// TIA Portal V20 export
// export: Created 2025-12-01T14:57:12.7432342Z, ExportSetting None, DisplayName Totally Integrated Automation Portal, DisplayVersion V20 Update 3, DisplayName TIA Portal Openness, DisplayVersion V20 Update 3, DisplayName TIA Portal Version Control Interface, DisplayVersion V20 Update 3, DisplayName STEP 7 Professional, DisplayVersion V20 Update 3, DisplayName STEP 7 Safety, DisplayVersion V20 Update 2, DisplayName WinCC Basic/Comfort/Advanced, DisplayVersion V20 Update 3, DisplayName WinCC Professional, DisplayVersion V20 Update 3, DisplayName WinCC Unified, DisplayVersion V20 Update 3
FUNCTION "FC756_EventosEstadoProcesoMaquina" : Void   // FC756, STL
TITLE = Emision de los Eventos del Proceso de la Maquina
{ S7_Optimized_Access := 'FALSE' }
AUTHOR : TRACKING
NAME : 20141014
VERSION : 4.0
// stored: AutoNumber false
   VAR_INPUT
      NumMaquina : UInt;   // Numero de Maquina
      EstadoMaquina : "EstadoZona";   // Estado de la Maquina
      EstadoVIMaquina : "EstadoMaquina";   // Estado del VI de la Maquina
      EmpezandoProceso : Bool;   // Aviso de Empezando el Proceso
      FinalProceso : Bool;   // Aviso de Final del Proceso
      ErrorProceso : Bool;   // Aviso de Error de Proceso
      MesaDeJDT02 : Bool;
   END_VAR
   VAR_TEMP
      NumeroUT : UInt;
      ProcesoActual : UInt;
      P_EmiEventos : DWord;
      DBEventos : Word;
      NumDBEventos : UInt;
      MaxBytes : UInt;
      NumBytes : UInt;
      OffsetInicial : UInt;
      OffsetFinal : UInt;
      Conversion : DWord;
      Convertir : UInt;
      Valor : UDInt;
   END_VAR
BEGIN

NETWORK
TITLE = Inicializaciones
///////////////////////////////////////////////////////////////////////////////
/// Inicio --> Pertenece al JDT 02

      L     "JDT1_NDB_EventosEmi";
      T     #DBEventos;
      T     #NumDBEventos;
      L     "JDT1_MaxBytes";
      T     #MaxBytes;

      AN    #MesaDeJDT02;
      JC    NoJdT02;

      L     "JDT2_NDB_EventosEmi";
      T     #DBEventos;
      T     #NumDBEventos;
      L     "JDT2_MaxBytes";
      T     #MaxBytes;

NoJdT02:NOP   0;

/// Final --> Pertenece al JDT 02
///////////////////////////////////////////////////////////////////////////////



NETWORK
TITLE = Mirar si se pueden generar eventos
// - Inicializo el Numero de Bytes y el puntero del DB de Eventos Generados
// - Calcula el Tamaño de bytes que hay en el DB de Eventos Genardos
// - Comprobamos si hay sitio para Eventos
///////////////////////////////////////////////////////////////////////////////
// Inicializo el Numero de Bytes y el puntero del DB Eventos Generados

      L     0;
      T     #NumBytes;  // Inicializo el numero de Bytes
      LAR2;  // Inicializo el puntero de Eventos Generados

///////////////////////////////////////////////////////////////////////////////
// Calcula el tamaño de bytes que hay en el DB Eventos Generados

      OPN   DB [#DBEventos];

Inicio_BusquedaFinalEventos:NOP   0;
      L     DBB [AR2, P#0.0];
      L     0;
      ==I;
      JC    Final_BusquedaFinalEventos;  // Buscamos el final del DB = 0

      +AR2  P#1.0;
      JU    Inicio_BusquedaFinalEventos;

Final_BusquedaFinalEventos:NOP   0;
      TAR2;  // Guardo el puntero
      T     #P_EmiEventos;  // Sacamos el NumBytes Escritos
      SRD   3;
      T     #NumBytes;

// -----------------------------------------------------------------------------------------------
// Comprobamos si hay sitio para mas Eventos

      L     #NumBytes;  // Miramos si hay sitio
      L     #MaxBytes;  // Max. que se pueden emitir, parametro
      >I;
      JC    Final;  // No se pueden generar más eventos



NETWORK
TITLE = Distribucion
///////////////////////////////////////////////////////////////////////////////
// --- Distribucion  del Estado del Proceso de la Maquina

      L     0;
      T     #ProcesoActual;

// ---------- Mirar si el Proceso esta Empezando

      A     #EmpezandoProceso;
      AN    #FinalProceso;
      AN    #ErrorProceso;
      JCN   _ST1;  // No Esta Empezando ?

      L     1011;  // Esta Empezando
      T     #ProcesoActual;
      JU    _STF;


// ---------- Mirar si el Proceso ha Finalizado

_ST1: AN    #EmpezandoProceso;
      A     #FinalProceso;
      AN    #ErrorProceso;
      JCN   _ST2;  // No Esta Finalizado ?

      L     1012;  // Esta Finalizado
      T     #ProcesoActual;
      JU    _STF;


// ---------- Mirar si el Proceso esta en Error

_ST2: AN    #EmpezandoProceso;
      AN    #FinalProceso;
      A     #ErrorProceso;
      JCN   _ST3;  // No Esta En Error ?

      L     1013;  // Esta En Error
      T     #ProcesoActual;
      JU    _STF;


// ---------- No se sabe como esta el Proceso

_ST3: L     0;  // No se Sabe
      T     "DB832_Maquinas".Maquinas[#NumMaquina].MemoriaEstado;  // Guardo como Nuevo

      JU    ST_F;


///////////////////////////////////////////////////////////////////////////////
// ---------- Mirar si hay que Emitir el Evento

_STF: NOP   0;
      L     "DB832_Maquinas".Maquinas[#NumMaquina].MemoriaEstado;
      L     #ProcesoActual;
      ==I;
      JC    ST_F;  // No ha cambio de Proceso ?

      L     0;
      L     #ProcesoActual;
      ==I;
      JC    ST_F;  // Y no sea Indetermiado ?

      JU    EmitirEvento;


///////////////////////////////////////////////////////////////////////////////
// --- Fin del Control

ST_F: JU    Final;



NETWORK
TITLE = Emision del Evento
EmitirEvento:NOP   0;

///////////////////////////////////////////////////////////////////////////////
// --- Formateo del Evento PROC - Estado del Proceso de la Maquina

      L     #P_EmiEventos;
      LAR2;  // Puntero al DB de Eventos Generados

      TAR2;  // Mirar si es el primer evento de la lista
      L     0;
      ==I;
      JC    NoEsInicio_ListaDeEventos;  // Es el primero

      OPN   DB [#DBEventos];
      L     ',';  // Separador entre eventos ','
      T     DBB [AR2, P#0.0];
      +AR2  P#1.0;

NoEsInicio_ListaDeEventos:NOP   0;
      OPN   DB [#DBEventos];  // DB de Eventos Generados (A Emitir)
      L     '{';  // Inicio de Evento '{'
      T     DBB [AR2, P#0.0];
      +AR2  P#1.0;


///////////////////////////////////////////////////////////////////////////////
// --- Cuerpo del Evento PROC

      L     'DATO';  // Evento 'DATO'
      T     DBD [AR2, P#0.0];
      +AR2  P#4.0;

      L     '[';  // Evento - Atributo Proceso '[PROC]'
      T     DBB [AR2, P#0.0];
      L     'PROC';
      T     DBD [AR2, P#1.0];
      L     ']';
      T     DBB [AR2, P#5.0];
      +AR2  P#6.0;

      L     "DB850_DefinicionMesas".Mesa[#NumMaquina].ConfigMesa.TipoMaquina;
      T     #Convertir;

      CALL  "FC895_Obtener_EtiquetaDeValor"
      ( ValorEvento    := #Convertir,
        EtiquetaEvento := #Conversion
      );

      OPN   DB [#DBEventos];
      L     #Conversion;
      T     DBD [AR2, P#0.0];
      +AR2  P#4.0;

      L     '[';  // Evento - Atributo MCKY '[MCKY]'
      T     DBB [AR2, P#0.0];
      L     'MCKY';
      T     DBD [AR2, P#1.0];
      L     ']';
      T     DBB [AR2, P#5.0];
      +AR2  P#6.0;

      TAR2;  // Guardar el Puntero
      T     #P_EmiEventos;  // Al DB de Eventos Generados

// --- Obtener Numero de McKey

      L     "DB810_ColasMesas".Colas[#NumMaquina].UT_PrimeraMesa;
      T     #NumeroUT;

      L     "DB812_UTs_Control".UT[#NumeroUT].Mckey;
      T     #Valor;

// --- Fin de Obtener el Mckey

      L     #P_EmiEventos;  // Recuperar el Puntero
      LAR2;  // Al DB de Eventos Generados

// --- Convertir Valor a ASCII - Mckey
      TAR2;
      SRD   3;
      T     #OffsetInicial;  // Miro que offset tiene la String

      CALL  "FC893_Obtener_StringDelAtributo"
      ( DB_String := #NumDBEventos,
        OffsetIni := #OffsetInicial,
        Valor     := #Valor,
        OffsetFin := #OffsetFinal
      );  // Llamo a ObtenerStrinAtributo

      L     #OffsetFinal;
      SLD   3;
      LAR2;  // Recupero que offset tiene la String

// --- Ya esta convertido el Valor a ASCI - Fin Mckey

      OPN   DB [#DBEventos];  // DB de Eventos Generados (A Emitir)
      L     '[';  // Evento - Atributo MESA '[MESA]'
      T     DBB [AR2, P#0.0];
      L     'MESA';
      T     DBD [AR2, P#1.0];
      L     ']';
      T     DBB [AR2, P#5.0];
      +AR2  P#6.0;

// --- Convertir Valor a ASCII - Numero de Mesa
      TAR2;
      SRD   3;
      T     #OffsetInicial;  // Miro que offset tiene la String

      L     "CTE_OffsetMesa";
      L     #NumMaquina;  // Numero de Maquina
      +I;
      T     #Valor;

      CALL  "FC893_Obtener_StringDelAtributo"
      ( DB_String := #NumDBEventos,
        OffsetIni := #OffsetInicial,
        Valor     := #Valor,
        OffsetFin := #OffsetFinal
      );  // Llamo a ObtenerStrinAtributo

      L     #OffsetFinal;
      SLD   3;
      LAR2;  // Recupero que offset tiene la String

// --- Ya esta convertido el Valor a ASCI - Numero de Mesa

      OPN   DB [#DBEventos];  // DB de Eventos Generados (A Emitir)
      L     '[';  // Evento - Atributo Resultado '[RSLT]'
      T     DBB [AR2, P#0.0];
      L     'RSLT';
      T     DBD [AR2, P#1.0];
      L     ']';
      T     DBB [AR2, P#5.0];
      +AR2  P#6.0;

      L     #ProcesoActual;
      T     #Convertir;  // Proceso _INI o _FIN o ERRO

      CALL  "FC895_Obtener_EtiquetaDeValor"
      ( ValorEvento    := #Convertir,
        EtiquetaEvento := #Conversion
      );

      OPN   DB [#DBEventos];  // DB de Eventos Generados (A Emitir)
      L     #Conversion;
      T     DBD [AR2, P#0.0];
      +AR2  P#4.0;


///////////////////////////////////////////////////////////////////////////////
// --- Final del formateo del Evento

      OPN   DB [#DBEventos];  // DB de Eventos Generados (A Emitir)
      L     '}';  // Fin de Evento '}'
      T     DBB [AR2, P#0.0];
      +AR2  P#1.0;

///////////////////////////////////////////////////////////////////////////////
// --- Dar por formateado el Evento

      L     #ProcesoActual;  // Lo doy por tratado
      T     "DB832_Maquinas".Maquinas[#NumMaquina].MemoriaEstado;

      JU    Final;  // Ya se ha generado el evento de la Maquina

// --- Fin del Formateo del Evento de Estado del Proceso
///////////////////////////////////////////////////////////////////////////////



NETWORK
TITLE = Fin de la Funcion
///////////////////////////////////////////////////////////////////////////////
//// -- Final de la Funcion
Final:NOP   0;



END_FUNCTION
